// TwinCAT 3 PLC project Untitled1
// ProgramVersion: 3.1.4023.0
// libraries:
//   Tc2_Standard, * (Beckhoff Automation GmbH)
//   Tc2_System, * (Beckhoff Automation GmbH)
//   Tc3_Module, * (Beckhoff Automation GmbH)
// project tree:
//   GVLs/ GVL.TcGVL
//   / PlcTask.TcTTO (not stored)
//   POUs/ FB_SOLVEXY.TcPOU, MAIN.TcPOU
// real-time tasks:
//   TASK PlcTask: cycle T#10ms, priority 20, ADS port 350
// I/O:
//   DEVICE Device 1 (EtherCAT), AmsNetId 5.72.137.238.2.1
//     Term 1 (EK1200) [EK1200-5000 EtherCAT Power supply (2A E-Bus)]
//       Term 2 (EL2004) [EL2004 4Ch. Dig. Output 24V, 0.5A]
//       Term 3 (EL2004) [EL2004 4Ch. Dig. Output 24V, 0.5A]
//       Term 4 (EL9011) [EL9011 End Terminal]

// ---- GVLs/GVL.TcGVL
{attribute 'qualified_only'}
VAR_GLOBAL
	
blink : BOOL := 1;


// Geometría del robot//
//todo en mm//

Pi : REAL := 3.1416;

d : REAL := 200;
l1 : REAL := 1000; //longitud brazo proximal
l2 : REAL := 1000; //longitud brazo distal

Xc : REAL:= 0; //posición x del spray
Yc : REAL:= 0; //posición y del spray

alfa : REAL:= Pi; //ángulo del brazo pxosimal izquierdo
beta : REAL:= 0; //ángulo del brazo pxosimal derecho

END_VAR

// ---- POUs/FB_SOLVEXY.TcPOU
FUNCTION_BLOCK FB_SOLVEXY
VAR_INPUT
x : REAL;
y : REAL;
END_VAR
VAR_OUTPUT
alfa : REAL;
beta : REAL;
END_VAR
VAR
END_VAR

alfa := ATAN(y/(GVL.d-x)) + ACOS ( (y*y + (x-GVL.d)*(x-GVL.d) + GVL.l1*GVL.l1 - GVL.l2*GVL.l2 ) / ( 2*GVL.l1*GVL.l2) );
beta := GVL.Pi - ATAN(y/(x-GVL.d)) - ACOS ( (y*y + (x-GVL.d)*(x-GVL.d) + GVL.l1*GVL.l1 - GVL.l2*GVL.l2 ) / ( 2*GVL.l1*GVL.l2) );

END_FUNCTION_BLOCK

// ---- POUs/MAIN.TcPOU
PROGRAM MAIN
VAR
	
fb_solvexy:FB_SOLVEXY;

END_VAR

GVL.blink := NOT(GVL.blink);

fb_solvexy.x:=GVL.Xc;
fb_solvexy.y:=GVL.Yc;
fb_solvexy();
GVL.alfa:=fb_solvexy.alfa;
GVL.beta:=fb_solvexy.beta;

END_PROGRAM
